(* PLC project OOP_Curso, Beckhoff Automation GmbH TwinCAT PLC Control 3.5.13.21 *)
(* stored: creationDateTime 2023-02-11T19:56:38.4759695, modificationDateTime 2023-02-11T19:56:38.480848 *)

(* global variable list GVL4 *)
//{attribute 'qualified_only'}
VAR_GLOBAL
	 nVarExt1 : INT; // 1st external variable
END_VAR

FUNCTION_BLOCK fb_tipos_de_datos
VAR_INPUT
	binput : BOOL;
END_VAR
VAR_INPUT
	binput2 : BOOL;
END_VAR
VAR_OUTPUT
	output1 : REAL;
END_VAR
VAR_IN_OUT
	in_out1 : LINT;
END_VAR
VAR_IN_OUT CONSTANT
	in_out_constant1 : DINT;
END_VAR
VAR
	var1 : STRING;
END_VAR
VAR_TEMP
	temp1 : ULINT;
END_VAR
VAR_STAT
    nVarStat1 : INT;
END_VAR
VAR_EXTERNAL
    nVarExt1 : INT; // 1st external variable
END_VAR
VAR PERSISTENT
    nVarPers1 : DINT; (* 1. Persistent variable *)
    bVarPers2 : BOOL; (* 2. Persistent variable *)
END_VAR
VAR RETAIN
    nRem1 : INT;
END_VAR
VAR CONSTANT
	n : INT:= 10;
END_VAR

            
          
END_FUNCTION_BLOCK

PROGRAM _04_Clases_y_Objetos
VAR
	fb :fb_tipos_de_datos;
	binput : BOOL;
	in_out1 : LINT;
	in_out_constant1 : DINT := 10;
END_VAR

            
fb(
//	binput:= binput, 
//	binput2:= , 
//	output1=> , 
	in_out1:= in_out1, 
	in_out_constant1:= in_out_constant1 );
          
END_PROGRAM
